// Mitsubishi GX Works2 project: PID_fx2n_funksjonstest_rykkfri   PLC: FX2N/FX2NC

// global labels: Global1
VAR_GLOBAL
  lampe_0 AT Y000 : BOOL;
  lampe_1 AT Y001 : BOOL;
  lampeVar_0 AT M100 : BOOL;
  lampeVar_1 AT M101 : BOOL;
  slider AT D0 : INT;
  tank AT D1 : INT;
  Input_KpValue AT D218 : REAL;  (* Valg av Kp verdi *)
  Input_TiValue AT D220 : REAL;  (* Valge av Ti verdi *)
  Input_TdValue AT D222 : REAL;  (* Valg av Td verdi *)
  Input_NValue AT D224 : REAL;  (* Valg av N verdi *)
  Input_TtValue AT D226 : REAL;  (* Valg av Tt verdi *)
  Input_AI_Raw AT D400 : INT;
  Output_AO_Raw AT D402 : INT;
  Input_ManualMode AT M500 : BOOL;  (* Valg av Manuell "1" eller Auto "0" *)
  Input_OperationModus AT M501 : BOOL;  (* Valg av direkte "1" eller Revers "0" Regulering *)
  Input_IntegratorModus AT M502 : BOOL;  (* Valg av Integrator virkning på regulator *)
  Input_DerivatorModus AT M503 : BOOL;  (* Valg av Derivator virkning på regulator *)
  Input_SamplingsTime AT D200 : INT;  (* Samplingstid sendt til PID *)
  Output_PID AT D202 : REAL;  (* Utgangs signal sendt ut fra PID *)
  Input_Referance AT D204 : REAL;  (* Referanse verdi sendt til PID *)
  Input_Process AT D206 : REAL;  (* Prosess verdi Sendt til PID *)
  Input_ManualValue AT D208 : REAL;  (* Manuell verdi sendt til PID *)
  Input_NomValue AT D210 : REAL;  (* Nominelt pådrag *)
  Input_MaxPådrag AT D212 : REAL;  (* Max pådrag *)
  Input_MinPådrag AT D214 : REAL;  (* Min pådrag *)
  Input_Skalert_Samplingstid AT D216 : ARRAY [0..1] OF INT;  (* Samplingstid skalert til timer *)
  Input_FF_TtValue AT D228 : REAL;  (* Valg av Tt verdi til LeadLag blokk *)
  Input_FF_TnValue AT D230 : REAL;  (* Valg av Tn verdi til LeadLag blokk *)
  Input_FF_KLLValue AT D232 : REAL;  (* Valg av KLL verdi til LeadLag blokk *)
  Output_Leadlag AT D234 : REAL;  (* Utgangsignal sendt ut fra LeadLag blokk *)
  Output_Total AT D236 : REAL;  (* Totalt utgangsignal summert *)
  Input_ErrorValue AT D238 : REAL;  (* Beregnet avvik *)
END_VAR

// task Task_01 (event TRUE, interval 0, priority 31): POU_01

PROGRAM POU_01
VAR
  LeadLag_1 : LeadLag;
  Output_Adder_1 : Output_Adder;
  My_PID_1 : My_PID;
END_VAR
(* structured ladder/FBD written out as ST: instructions are called as NAME(EN, inputs, outputs); _pN, _eN, _tN stand for wires *)
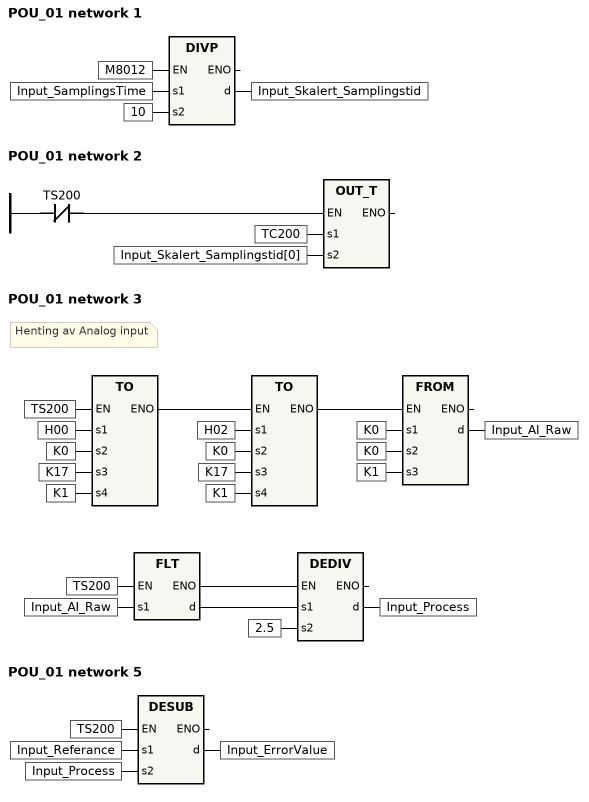
(* network 1 *)
DIVP(M8012, Input_SamplingsTime, 10, Input_Skalert_Samplingstid);
(* network 2 *)
OUT_T(NOT TS200, TC200, Input_Skalert_Samplingstid[0]);
(* network 3 *)
(* Henting av Analog input *)
_e1 := TO(TS200, H00, K0, K17, K1);
_e2 := TO(_e1, H02, K0, K17, K1);
FROM(_e2, K0, K0, K1, Input_AI_Raw);
_e4 := FLT(TS200, Input_AI_Raw, _t3);
DEDIV(_e4, _t3, 2.5, Input_Process);
(* network 5 *)
DESUB(TS200, Input_Referance, Input_Process, Input_ErrorValue);
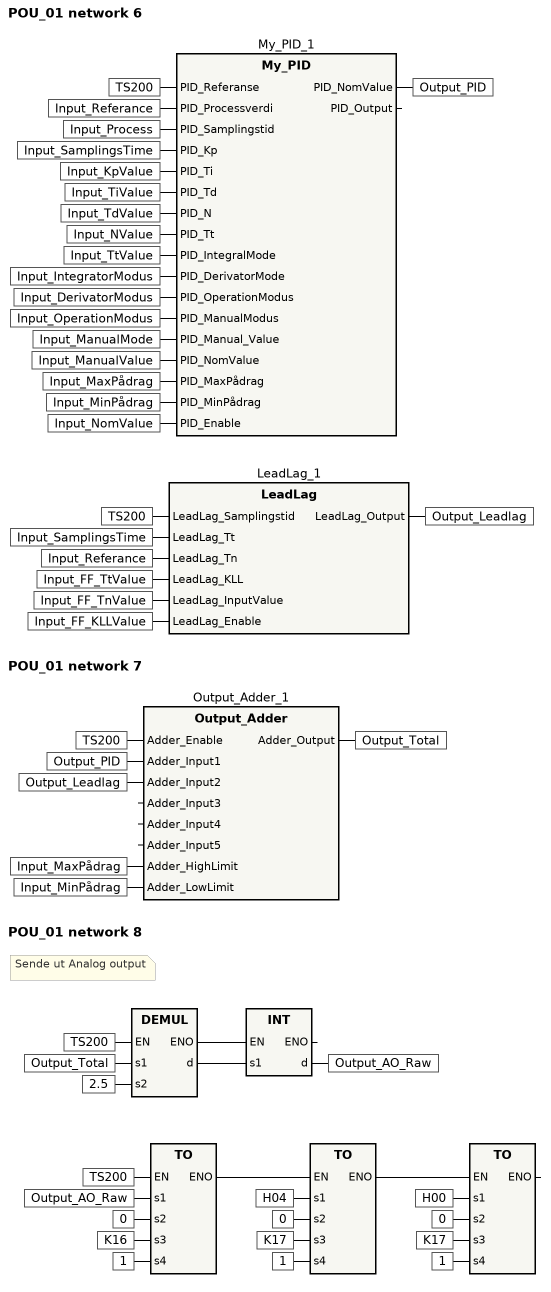
(* network 6 *)
My_PID_1(PID_Referanse := TS200, PID_Processverdi := Input_Referance, PID_Samplingstid := Input_Process, PID_Kp := Input_SamplingsTime, PID_Ti := Input_KpValue, PID_Td := Input_TiValue, PID_N := Input_TdValue, PID_Tt := Input_NValue, PID_IntegralMode := Input_TtValue, PID_DerivatorMode := Input_IntegratorModus, PID_OperationModus := Input_DerivatorModus, PID_ManualModus := Input_OperationModus, PID_Manual_Value := Input_ManualMode, PID_NomValue := Input_ManualValue, PID_MaxPådrag := Input_MaxPådrag, PID_MinPådrag := Input_MinPådrag, PID_Enable := Input_NomValue);
Output_PID := My_PID_1.PID_NomValue;
LeadLag_1(LeadLag_Samplingstid := TS200, LeadLag_Tt := Input_SamplingsTime, LeadLag_Tn := Input_Referance, LeadLag_KLL := Input_FF_TtValue, LeadLag_InputValue := Input_FF_TnValue, LeadLag_Enable := Input_FF_KLLValue, LeadLag_Output => Output_Leadlag);
(* network 7 *)
Output_Adder_1(Adder_Enable := TS200, Adder_Input1 := Output_PID, Adder_Input2 := Output_Leadlag, Adder_HighLimit := Input_MaxPådrag, Adder_LowLimit := Input_MinPådrag, Adder_Output => Output_Total);
(* network 8 *)
(* Sende ut Analog output *)
_e2 := DEMUL(TS200, Output_Total, 2.5, _t1);
INT(_e2, _t1, Output_AO_Raw);
_e3 := TO(TS200, Output_AO_Raw, 0, K16, 1);
_e4 := TO(_e3, H04, 0, K17, 1);
TO(_e4, H00, 0, K17, 1);
END_PROGRAM

FUNCTION_BLOCK My_PID
VAR_INPUT
  PID_Referanse : REAL;  (* Referanseverdi PID blokk *)
  PID_Processverdi : REAL;  (* Prosessverdi PID blokk *)
  PID_Samplingstid : INT;  (* Samplingstid PID blokk (ms) *)
  PID_Kp : REAL;  (* KP PID blokk *)
  PID_Ti : REAL;  (* Ti PID blokk *)
  PID_Td : REAL;  (* Td PID blokk *)
  PID_N : REAL;  (* Filter konstant for Tf *)
  PID_Tt : REAL;  (* Tracking konstant for PID tracking inngang *)
  PID_IntegralMode : BOOL;  (* Integrator for PID blokk *)
  PID_DerivatorMode : BOOL;  (* Derivator for PID blokk *)
  PID_OperationModus : BOOL;  (* Direkte kobling "1", reversert "0" *)
  PID_ManualModus : BOOL;  (* Auto "0" , Manuell pådrag "1" *)
  PID_Manual_Value : REAL;  (* Manuelt pådrag verdi *)
END_VAR
VAR_IN_OUT
  PID_NomValue : REAL;  (* Nominelt pådrags verdi *)
END_VAR
VAR_INPUT
  PID_MaxPådrag : REAL;  (* Max pådrags verdi *)
  PID_MinPådrag : REAL;  (* Min pådrags verdi *)
END_VAR
VAR_OUTPUT
  PID_Output : REAL;  (* Utgangsverdi fra PID-reg *)
END_VAR
VAR
  PID_Alpha : REAL;  (* Beregnet alpha verdi *)
  PID_Beta : REAL;  (* Beregnet betaverdi *)
  PID_Gamma : REAL;  (* Beregnet gammaverdi *)
  PID_ErrorValue_F : ARRAY [0..1] OF REAL;  (* Beregnet error verdi (Denne og forrige verdi) *)
  PID_PGain : ARRAY [0..1] OF REAL;  (* Beregnet P forsterkning (Denne og forrige verdi) *)
  PID_IGain : ARRAY [0..1] OF REAL;  (* Beregnet I forsterkning (Denne og forrige verdi) *)
  PID_DGain : ARRAY [0..1] OF REAL;  (* Beregnet D forsterkning (Denne og forrige verdi) *)
  PID_Gain_Total : REAL;  (* Beregnet sum av total pådrag (Ubegrenset verdi) *)
  PID_Gain_Tracking : REAL;  (* Beregnet sum av tracking pådrag (Begrenset verdi) *)
  PID_Processverdi_F : ARRAY [0..1] OF REAL;  (* Prosess verdi i PID blokk (denne og forrige verdi) *)
  PID_Skalert_Samplingstid : REAL;  (* Skalert samplingstid i sekunder *)
  PID_Mellomregning_Samplingstid : REAL;  (* Mellomregning av samplingstid *)
END_VAR
VAR_INPUT
  PID_Enable : BOOL;  (* Samplings enable *)
END_VAR
VAR
  Regulatortype : ARRAY [0..1] OF INT;  (* Array to know current and last regulator type *)
  tiss : REAL;
END_VAR
(*Omgjøring av samplingstid fra ms til s*)
FLT(TRUE , PID_Samplingstid, PID_Mellomregning_Samplingstid);
PID_Skalert_Samplingstid := PID_Mellomregning_Samplingstid/1000.0;



(*Systemet vil gå inn i koden hvert samplingstid som er satt*)

IF PID_Enable THEN	
	(*Regning av konstanter alpha, beta og omgjøring av prosess, nominelt-, min og max pådrag og ref verdi til float*)
	PID_Alpha := PID_Skalert_Samplingstid/PID_Ti;
    PID_Beta := PID_Td/(PID_Td + (PID_Skalert_Samplingstid*pid_n));
	PID_Processverdi_F[0] := PID_Processverdi;
	IF PID_Tt > 0.0 THEN 
		PID_Gamma:= PID_Skalert_Samplingstid/PID_Tt;
	ELSE
		PID_Gamma:= 0.0;
	END_IF;

	(*IF statement to differentiate between the regulator types:		0 = P-reg.	1 = PD-reg.	2 = PI-reg.	3 = PID-reg*)
	IF PID_IntegralMode AND PID_DerivatorMode THEN
		Regulatortype[0] := 3; (*PID-regulator*)													
	ELSIF PID_IntegralMode AND NOT PID_DerivatorMode THEN
		Regulatortype[0] := 2; (*PI-regulator*)
	ELSIF PID_DerivatorMode AND NOT PID_IntegralMode THEN
		Regulatortype[0] := 1; (*PD-regulator*)
	ELSE
		Regulatortype[0] := 0; (*P-regulator*) 
	END_IF;
	
	(*IF statement that sets PID_IGain[0] to PID_NomValue if switching from P to PI or PID reg. when nominal value is not 0.0, and PID_IGain[0] to 0.0 if switching from P to PI or PID reg. when nominal value = 0.0.*)
	(*This prevents leaps in the PID_output value when switching to a regulator with integral gain.*)
	IF PID_NomValue <> 0.0 AND Regulatortype[0] = 2 AND Regulatortype[1] = 0 OR PID_NomValue <> 0.0 AND Regulatortype[0] = 3 AND Regulatortype[1] = 0 THEN
		PID_IGain[0] := PID_NomValue;
	ELSIF PID_NomValue = 0.0 AND Regulatortype[0] = 2 AND Regulatortype[1] = 0 OR  PID_NomValue = 0.0 AND Regulatortype[0] = 3 AND Regulatortype[1] = 0 THEN
		PID_IGain[0] := 0.0;
	END_IF;
	
	(*IF statement that sets PID_IGain[0] to PID_NomValue if switching from PD to PI or PID reg. when nominal value is not 0.0, and PID_IGain[0] to 0.0 if switching from PD to PI or PID reg. when nominal value = 0.0.*)
	(*This prevents leaps in the PID_output value when switching to a regulator with integral gain.*)
	IF PID_NomValue <> 0.0 AND Regulatortype[0] = 2 AND Regulatortype[1] = 1 OR PID_NomValue <> 0.0 AND Regulatortype[0] = 3 AND Regulatortype[1] = 1 THEN
		PID_IGain[0] := PID_NomValue;
	ELSIF PID_NomValue = 0.0 AND Regulatortype[0] = 2 AND Regulatortype[1] = 1 OR  PID_NomValue = 0.0 AND Regulatortype[0] = 3 AND Regulatortype[1] = 1 THEN
		PID_IGain[0] := 0.0;
	END_IF;
	
	(*IF statement that prevents leaps in the PID_output value when sitching to a regulator without integral gain*)
	IF Regulatortype[0] = 0 AND Regulatortype[1] = 2 OR  Regulatortype[0] = 0 AND Regulatortype[1] = 3 THEN
		PID_NomValue:= PID_IGain[0]+PID_NomValue;
	END_IF;
	
	(*IF statement that prevents leaps in the PID_output value when sitching to a regulator without integral gain*)
	IF Regulatortype[0] = 1 AND Regulatortype[1] = 2 OR  Regulatortype[0] = 1 AND Regulatortype[1] = 3 THEN
		PID_NomValue:= PID_IGain[0]+PID_NomValue;
	END_IF;
	
	(*Leaps in the PID_output value when sitching to a regulator with derivative gain is prevented by swithing when the system is stable. Same is applicaple when switching to a regulator without derivative gain.*)
	
	Regulatortype[1] := Regulatortype[0]; (*Last regulator type stored in variable*)
	
	(*Regning av avvik mtp om det er direkte eller revers regulering*)
	IF PID_OperationModus THEN
		PID_ErrorValue_F[0] := PID_Processverdi_F[0] - PID_Referanse;
	ELSE
		PID_ErrorValue_F[0] := PID_Referanse - PID_Processverdi_F[0];
	END_IF;
	

	(*Beregning av pådragsbidrag fra P-del*)
	PID_PGain[0] := PID_Kp*PID_ErrorValue_F[0];
	
	
	(*Ser om integrator er aktivert og beregner pådragsbidrag fra I-del med tracking inngang*)
	IF PID_IntegralMode  THEN
		PID_IGain[0] := PID_IGain[1] + PID_Kp*PID_Alpha*PID_ErrorValue_F[0]+PID_Gamma*(PID_Gain_Tracking-PID_Gain_Total);
	
	ELSE
		PID_IGain[0] := 0.0;
	END_IF;
	
	
	(*Ser om Derivator er aktivert og beregner pådragsbidrag fra D-del*)
	IF PID_DerivatorMode THEN
		PID_DGain[0] := (PID_Beta*PID_DGain[1]) - ((PID_Kp*PID_Td/PID_Skalert_Samplingstid)*(1.0-PID_Beta)*(PID_Processverdi_F[0]-PID_Processverdi_F[1]));
	ELSE 
		PID_DGain[0] := 0.0;
	END_IF;
	
	(*Summerer sammen pådragsbidrag fra alle delene*)
	PID_Gain_Total := PID_PGain[0] + PID_IGain[0] + PID_DGain[0] + PID_NomValue;
	
	(*Oppdatering av verdier*)
	PID_ErrorValue_F[1] := PID_ErrorValue_F[0];
	PID_Processverdi_F[1] := PID_Processverdi_F[0];
	PID_PGain[1] := PID_PGain[0];
	PID_IGain[1] := PID_IGain[0];
	PID_DGain[1] := PID_DGain[0];
	
	IF PID_ManualModus THEN 
		(*Kontrollerer at manuelt pådrag er innenfor min og max verdi*)
		PID_Gain_Tracking := PID_Manual_Value;
	ELSE 
		PID_Gain_Tracking := PID_Gain_Total;
	END_IF;
	
		(*Kontrollerer at pådragsbidrag er innenfor min og max verdier*)
	IF PID_Gain_Tracking > PID_MaxPådrag THEN
		PID_Gain_Tracking:= PID_MaxPådrag ;
	ELSIF PID_Gain_Tracking< PID_MinPådrag THEN 
		PID_Gain_Tracking:= PID_MinPådrag;
	ELSE
		PID_Gain_Tracking:= PID_Gain_Tracking;
	END_IF;


		
	(*Utgang fra PID regulator*)
	PID_Output := PID_Gain_Tracking;
ELSE 
	PID_Output:= PID_Gain_Tracking;
END_IF;
END_FUNCTION_BLOCK

FUNCTION_BLOCK LeadLag
VAR_INPUT
  LeadLag_Samplingstid : INT;  (* Samplingstid Lead Lag blokk *)
  LeadLag_Tt : REAL;  (* Tt konstant for Lead Lag blokk *)
  LeadLag_Tn : REAL;  (* Tn konstant for Lead Lag blokk *)
  LeadLag_KLL : REAL;  (* KLL konstant for Lead Lag blokk *)
END_VAR
VAR
  LeadLag_Mellomregning_Sampl : REAL;  (* Mellom regning for samplingstid *)
  LeadLag_Skalert_Samplingstid : REAL;  (* Skalert samplingstid i sekunder *)
END_VAR
VAR_INPUT
  LeadLag_InputValue : REAL;  (* Inngangsverdi inn til LeadLag blokk *)
END_VAR
VAR
  LeadLag_InputValue_F : ARRAY [0..1] OF REAL;  (* Input verdi denne og forrige *)
  LeadLag_Output_F : ARRAY [0..1] OF REAL;  (* Utgangspådrag  (denne og forrige) *)
END_VAR
VAR_OUTPUT
  LeadLag_Output : REAL;  (* Utgangsverdu ut fra LeadLag blokk *)
END_VAR
VAR_INPUT
  LeadLag_Enable : BOOL;  (* Enable for hvert samplingstid *)
END_VAR
(*Omgjøring av samplingstid fra ms til s*)
FLT(TRUE , leadlag_Samplingstid, leadLag_Mellomregning_Sampl);
LeadLag_Skalert_Samplingstid := leadlag_Mellomregning_Sampl/1000.0;

IF LeadLag_Enable THEN
	LeadLag_InputValue_F[0] := LeadLag_InputValue;
	
	LeadLag_Output_F[0] := (LeadLag_KLL*((LeadLag_Tt+LeadLag_Skalert_Samplingstid)*LeadLag_InputValue_F[0]-LeadLag_Tt*LeadLag_InputValue_F[1])+LeadLag_Tn*LeadLag_Output_F[1])/(LeadLag_Tn+LeadLag_Skalert_Samplingstid);
	
	LeadLag_Output_F[1] := LeadLag_Output_F[0];
	LeadLag_InputValue_F[1] := LeadLag_InputValue_F[0];
	
	LeadLag_Output := LeadLag_Output_F[0];
ELSE

;
END_IF;


;
END_FUNCTION_BLOCK

FUNCTION_BLOCK Output_Adder
VAR_INPUT
  Adder_Enable : BOOL;
  Adder_Input1 : REAL;  (* Input value 1 *)
  Adder_Input2 : REAL;  (* Input value 2 *)
  Adder_Input3 : REAL;  (* Input value 3 *)
  Adder_Input4 : REAL;  (* Input value 4 *)
  Adder_Input5 : REAL;  (* Input value 5 *)
  Adder_HighLimit : REAL;  (* Maximum output *)
  Adder_LowLimit : REAL;  (* Minimum output *)
END_VAR
VAR_OUTPUT
  Adder_Output : REAL;  (* Total output from adder *)
END_VAR
VAR
  Adder_Sum : REAL;  (* Sum av inputs *)
END_VAR
IF Adder_Enable THEN
	Adder_Sum := Adder_Input1+Adder_Input2+Adder_Input3+Adder_Input4+Adder_Input5;
	
	IF Adder_Sum > Adder_HighLimit THEN
		Adder_Output := Adder_HighLimit;
	ELSIF Adder_Sum < Adder_LowLimit THEN
		Adder_Output := Adder_LowLimit;
	ELSE
		Adder_Output := Adder_Sum;
	END_IF;
END_IF;
;
END_FUNCTION_BLOCK
